{attribute 'GeneratedUsingTerminal: EK1122-0000-0018'}
{attribute addProperty BoxType "EK1122-0000-0018"}
{attribute addProperty Id "Beckhoff_AMI8xxxsub_EK1100EK1100_1FC0878B2A_0001_AMI8000_0000_0016AMI8000_68DB4BA039A_0002_AMI8000_0090_0016AMI8000_68DB4BA039"}
{attribute addProperty CRC "1921153808"}
{attribute addProperty Size "80"}
TYPE Beckhoff_AMI8xxxEK1122_72827B10 EXTENDS EK1122_1FC0878B :
STRUCT
	{attribute addProperty Name "Beckhoff AMI8xxxsub EK1100"}
	{attribute addProperty PreviousPort "Beckhoff AMI8xxxEK1122 : D"}
	Beckhoff_AMI8xxxsub_EK1100 : EK1100_1FC0878B;
	{attribute addProperty Name "A_0001(AMI8000-0000-0016)"}
	{attribute addProperty PreviousPort "Beckhoff AMI8xxxsub EK1100 : C"}
	A_0001_AMI8000_0000_0016 : AMI8000_68DB4BA0;
	{attribute addProperty Name "A_0002(AMI8000-0090-0016)"}
	{attribute addProperty PreviousPort "A_0001(AMI8000-0000-0016) : B"}
	A_0002_AMI8000_0090_0016 : AMI8000_68DB4BA0;
END_STRUCT
END_TYPE

(* stored: Version 1.2.0.0, ProductVersion 3.1.4024.11
   DUT Beckhoff_AMI8xxxEK1122_72827B10: Id {4c6a2afa-4175-4c8b-b29a-b6158de70981} *)
